TYPE ST_LogEntry :
STRUCT
	sSeverity		:  STRING( 24 );
	sSourceName		: T_MaxString;
	sTimestampLog	: STRING( 24 );
	MethodName		: STRING( 24 );
	sText			: T_MaxString;
END_STRUCT
END_TYPE

(* stored: Version 1.1.0.1, ProductVersion 3.1.4026.18
   DUT ST_LogEntry: Id {6cbe7644-ef16-4b20-872a-817412391647} *)
